{attribute 'qualified_only'}
{attribute 'strict'}
TYPE INTERNAL eCylinderStep :
(
    RESET,
    IN_HOME_POS,
    MOVE_TO_WORK_POS,
    IN_WORK_POS,
    MOVE_TO_HOME_POS,
    ERROR
);
END_TYPE

(* stored: Version 1.1.0.1, ProductVersion 3.1.4024.12
   DUT eCylinderStep: Id {75761d77-4adb-4813-9528-4a7a43006adb} *)
